// TIA Portal V20 export
DATA_BLOCK "ET200SP_205"   // DB274
// stored: MemoryReserve 100
   VAR
      "SP205.00 Main OP: pendant required on, yellow" : Bool;
      SPARE1 : Bool;
      "SP205.02 Main OP: home on, green" : Bool;
      SPARE2 : Bool;
      SPARE3 : Bool;
      SPARE4 : Bool;
      SPARE5 : Bool;
      "SP205.07 Main OP: SCS Disable mode selected, green" : Bool;
   END_VAR
BEGIN
END_DATA_BLOCK
